// TwinCAT 3 PLC project PLC
// ProgramVersion: 3.1.4024.0
// libraries:
//   Tc2_ControllerToolbox, * (Beckhoff Automation GmbH)
//   Tc2_Standard, * (Beckhoff Automation GmbH)
//   Tc2_System, * (Beckhoff Automation GmbH)
//   Tc3_Module, * (Beckhoff Automation GmbH)
// project tree:
//   / PlcTask.TcTTO
//   POUs/ MAIN.TcPOU
// real-time tasks:
//   TASK PlcTask: cycle T#13ms, priority 20, ADS port 350
// I/O:
//   DEVICE Device 2 (CX7000), AmsNetId 5.103.237.148.3.1
//     Term 1 (CX7028) [CX7028-0000-0121]
//       modules: Module 1 (DIO_2x), Module 2 (Empty Module), Module 3 (PWM_DI_2x), Module 4 (Empty Module), Module 5 (DI_2x), Module 6 (Empty Module), Module 7 (DI_2x), Module 8 (Empty Module)
// variable links:
//   PLC/PLC Instance <-> Device 2 (CX7000)/Term 1 (CX7028)
//     PlcTask Inputs/MAIN.bServoClosedSignal <-> Module 1 (DIO_2x)/DIO_2x Input Channel 1/Input
//     PlcTask Outputs/MAIN.iPWMOutput <-> Module 3 (PWM_DI_2x)/PWM_DI_2x Outputs Channel 1/PWM output
//     PlcTask Outputs/MAIN.iPWMPeriod <-> Module 3 (PWM_DI_2x)/PWM_DI_2x Outputs Channel 1/PWM period

CONFIGURATION PLC
    RESOURCE PLC ON TwinCAT3
        TASK PlcTask(INTERVAL := T#13ms, PRIORITY := 20);
        PROGRAM MAIN WITH PlcTask : MAIN;
    END_RESOURCE
END_CONFIGURATION

// ---- POUs/MAIN.TcPOU
PROGRAM MAIN
VAR
	// Close hand signal from output of C6032
	bServoClosedSignal AT %I*	:	BOOL;
	

	// PWM Controls
	iPWMOutput AT %Q*			:	UINT;
	iPWMPeriod AT %Q*			:	UINT;

END_VAR

iPWMPeriod := 10000;
IF bServoClosedSignal THEN
	iPWMOutput := 9000;
ELSE
	iPWMOutput := 3300;
END_IF

END_PROGRAM
